PROGRAM P3_00_MAIN
VAR
	tonDeleteDelay			:TON;
END_VAR

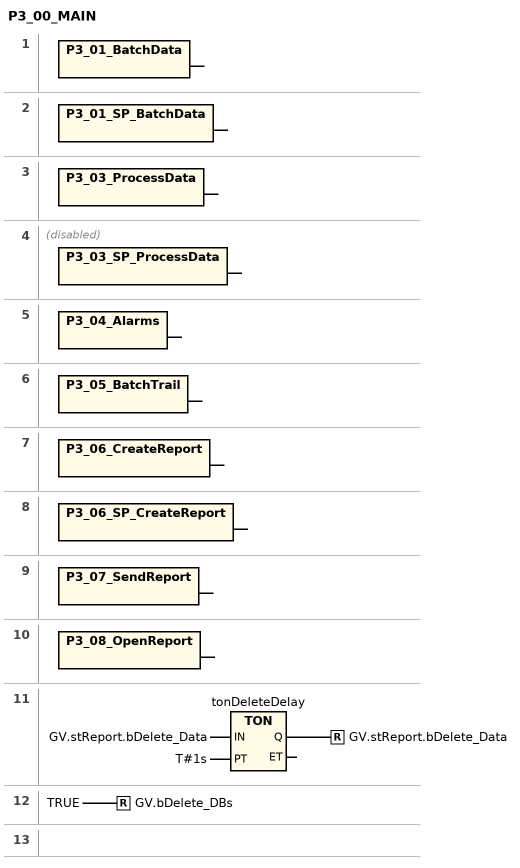
// NETWORK 1
P3_01_BatchData();

// NETWORK 2
P3_01_SP_BatchData();

// NETWORK 3
P3_03_ProcessData();

// NETWORK 4 (disabled)
// P3_03_SP_ProcessData();

// NETWORK 5
P3_04_Alarms();

// NETWORK 6
P3_05_BatchTrail();

// NETWORK 7
P3_06_CreateReport();

// NETWORK 8
P3_06_SP_CreateReport();

// NETWORK 9
P3_07_SendReport();

// NETWORK 10
P3_08_OpenReport();

// NETWORK 11
tonDeleteDelay(IN := GV.stReport.bDelete_Data, PT := T#1s); // TON
GV.stReport.bDelete_Data R= tonDeleteDelay.Q;

// NETWORK 12
GV.bDelete_DBs R= TRUE;

// NETWORK 13

END_PROGRAM

(* stored: Version 1.1.0.1, ProductVersion 3.1.4026.13
   POU P3_00_MAIN: Id {6dbcf589-6ccb-47fd-98a1-d1c85a02152b}, SpecialFunc None *)
